DATA_BLOCK "DB_HGU_Execution"
TITLE = 'HGU Execution Variables Data Block'
{ S7_Optimized_Access := 'TRUE' }
VERSION : 1.0
// =============================================================================
// TUSAŞ HGU Control System - Execution Variables Data Block
// TIA Portal S7-1500 Structured Control Language (SCL)
// Generated: 2025-01-14
// Description: All execution variables for HGU system synchronized with UI
// =============================================================================
   VAR
      MOTOR_1_RPM_EXECUTION : Real;   // Motor 1 RPM Execution Value
      MOTOR_1_CURRENT_EXECUTION : Real;   // Motor 1 Current (A) Execution Value
      MOTOR_1_TARGET_EXECUTION : Real;   // Motor 1 Target RPM Execution Value
      MOTOR_1_FLOW_EXECUTION : Real;   // Motor 1 Flow Rate (L/min) Execution Value
      MOTOR_1_PRESSURE_EXECUTION : Real;   // Motor 1 Pressure (bar) Execution Value
      MOTOR_1_LEAK_EXECUTION : Real;   // Motor 1 Leak Rate (L/min) Execution Value
      MOTOR_1_TEMPERATURE_EXECUTION : Real;   // Motor 1 Temperature (°C) Execution Value
      MOTOR_1_STATUS_EXECUTION : USInt;   // Motor 1 Status (0=Offline, 1=Ready, 2=Running, 3=Error)
      MOTOR_1_VALVE_EXECUTION : USInt;   // Motor 1 Valve Control (0=Closed, 1=Open)
      MOTOR_1_LINE_FILTER_EXECUTION : USInt;   // Motor 1 Line Filter Status (0=Error, 1=Warning, 2=OK)
      MOTOR_1_SUCTION_FILTER_EXECUTION : USInt;   // Motor 1 Suction Filter Status (0=Error, 1=OK)
      MOTOR_1_ENABLE_EXECUTION : Bool;   // Motor 1 Enable Control (FALSE=Disabled, TRUE=Enabled)
      MOTOR_1_FLOW_SETPOINT : Real;   // Motor 1 Flow Setpoint (L/min) - User Adjustable from Popup
      // Motor-Pump #2 Variables
      MOTOR_2_RPM_EXECUTION : Real;   // Motor 2 RPM Execution Value
      MOTOR_2_CURRENT_EXECUTION : Real;   // Motor 2 Current (A) Execution Value
      MOTOR_2_TARGET_EXECUTION : Real;   // Motor 2 Target RPM Execution Value
      MOTOR_2_FLOW_EXECUTION : Real;   // Motor 2 Flow Rate (L/min) Execution Value
      MOTOR_2_PRESSURE_EXECUTION : Real;   // Motor 2 Pressure (bar) Execution Value
      MOTOR_2_LEAK_EXECUTION : Real;   // Motor 2 Leak Rate (L/min) Execution Value
      MOTOR_2_TEMPERATURE_EXECUTION : Real;   // Motor 2 Temperature (°C) Execution Value
      MOTOR_2_STATUS_EXECUTION : USInt;   // Motor 2 Status (0=Offline, 1=Ready, 2=Running, 3=Error)
      MOTOR_2_VALVE_EXECUTION : USInt;   // Motor 2 Valve Control (0=Closed, 1=Open)
      MOTOR_2_LINE_FILTER_EXECUTION : USInt;   // Motor 2 Line Filter Status (0=Error, 1=Warning, 2=OK)
      MOTOR_2_SUCTION_FILTER_EXECUTION : USInt;   // Motor 2 Suction Filter Status (0=Error, 1=OK)
      MOTOR_2_ENABLE_EXECUTION : Bool;   // Motor 2 Enable Control (FALSE=Disabled, TRUE=Enabled)
      MOTOR_2_FLOW_SETPOINT : Real;   // Motor 2 Flow Setpoint (L/min) - User Adjustable from Popup
      // Motor-Pump #3 Variables
      MOTOR_3_RPM_EXECUTION : Real;   // Motor 3 RPM Execution Value
      MOTOR_3_CURRENT_EXECUTION : Real;   // Motor 3 Current (A) Execution Value
      MOTOR_3_TARGET_EXECUTION : Real;   // Motor 3 Target RPM Execution Value
      MOTOR_3_FLOW_EXECUTION : Real;   // Motor 3 Flow Rate (L/min) Execution Value
      MOTOR_3_PRESSURE_EXECUTION : Real;   // Motor 3 Pressure (bar) Execution Value
      MOTOR_3_LEAK_EXECUTION : Real;   // Motor 3 Leak Rate (L/min) Execution Value
      MOTOR_3_TEMPERATURE_EXECUTION : Real;   // Motor 3 Temperature (°C) Execution Value
      MOTOR_3_STATUS_EXECUTION : USInt;   // Motor 3 Status (0=Offline, 1=Ready, 2=Running, 3=Error)
      MOTOR_3_VALVE_EXECUTION : USInt;   // Motor 3 Valve Control (0=Closed, 1=Open)
      MOTOR_3_LINE_FILTER_EXECUTION : USInt;   // Motor 3 Line Filter Status (0=Error, 1=Warning, 2=OK)
      MOTOR_3_SUCTION_FILTER_EXECUTION : USInt;   // Motor 3 Suction Filter Status (0=Error, 1=OK)
      MOTOR_3_ENABLE_EXECUTION : Bool;   // Motor 3 Enable Control (FALSE=Disabled, TRUE=Enabled)
      MOTOR_3_FLOW_SETPOINT : Real;   // Motor 3 Flow Setpoint (L/min) - User Adjustable from Popup
      // Motor-Pump #4 Variables
      MOTOR_4_RPM_EXECUTION : Real;   // Motor 4 RPM Execution Value
      MOTOR_4_CURRENT_EXECUTION : Real;   // Motor 4 Current (A) Execution Value
      MOTOR_4_TARGET_EXECUTION : Real;   // Motor 4 Target RPM Execution Value
      MOTOR_4_FLOW_EXECUTION : Real;   // Motor 4 Flow Rate (L/min) Execution Value
      MOTOR_4_PRESSURE_EXECUTION : Real;   // Motor 4 Pressure (bar) Execution Value
      MOTOR_4_LEAK_EXECUTION : Real;   // Motor 4 Leak Rate (L/min) Execution Value
      MOTOR_4_TEMPERATURE_EXECUTION : Real;   // Motor 4 Temperature (°C) Execution Value
      MOTOR_4_STATUS_EXECUTION : USInt;   // Motor 4 Status (0=Offline, 1=Ready, 2=Running, 3=Error)
      MOTOR_4_VALVE_EXECUTION : USInt;   // Motor 4 Valve Control (0=Closed, 1=Open)
      MOTOR_4_LINE_FILTER_EXECUTION : USInt;   // Motor 4 Line Filter Status (0=Error, 1=Warning, 2=OK)
      MOTOR_4_SUCTION_FILTER_EXECUTION : USInt;   // Motor 4 Suction Filter Status (0=Error, 1=OK)
      MOTOR_4_ENABLE_EXECUTION : Bool;   // Motor 4 Enable Control (FALSE=Disabled, TRUE=Enabled)
      MOTOR_4_FLOW_SETPOINT : Real;   // Motor 4 Flow Setpoint (L/min) - User Adjustable from Popup
      // Motor-Pump #5 Variables
      MOTOR_5_RPM_EXECUTION : Real;   // Motor 5 RPM Execution Value
      MOTOR_5_CURRENT_EXECUTION : Real;   // Motor 5 Current (A) Execution Value
      MOTOR_5_TARGET_EXECUTION : Real;   // Motor 5 Target RPM Execution Value
      MOTOR_5_FLOW_EXECUTION : Real;   // Motor 5 Flow Rate (L/min) Execution Value
      MOTOR_5_PRESSURE_EXECUTION : Real;   // Motor 5 Pressure (bar) Execution Value
      MOTOR_5_LEAK_EXECUTION : Real;   // Motor 5 Leak Rate (L/min) Execution Value
      MOTOR_5_TEMPERATURE_EXECUTION : Real;   // Motor 5 Temperature (°C) Execution Value
      MOTOR_5_STATUS_EXECUTION : USInt;   // Motor 5 Status (0=Offline, 1=Ready, 2=Running, 3=Error)
      MOTOR_5_VALVE_EXECUTION : USInt;   // Motor 5 Valve Control (0=Closed, 1=Open)
      MOTOR_5_LINE_FILTER_EXECUTION : USInt;   // Motor 5 Line Filter Status (0=Error, 1=Warning, 2=OK)
      MOTOR_5_SUCTION_FILTER_EXECUTION : USInt;   // Motor 5 Suction Filter Status (0=Error, 1=OK)
      MOTOR_5_ENABLE_EXECUTION : Bool;   // Motor 5 Enable Control (FALSE=Disabled, TRUE=Enabled)
      MOTOR_5_FLOW_SETPOINT : Real;   // Motor 5 Flow Setpoint (L/min) - User Adjustable from Popup
      // Motor-Pump #6 Variables
      MOTOR_6_RPM_EXECUTION : Real;   // Motor 6 RPM Execution Value
      MOTOR_6_CURRENT_EXECUTION : Real;   // Motor 6 Current (A) Execution Value
      MOTOR_6_TARGET_EXECUTION : Real;   // Motor 6 Target RPM Execution Value
      MOTOR_6_FLOW_EXECUTION : Real;   // Motor 6 Flow Rate (L/min) Execution Value
      MOTOR_6_PRESSURE_EXECUTION : Real;   // Motor 6 Pressure (bar) Execution Value
      MOTOR_6_LEAK_EXECUTION : Real;   // Motor 6 Leak Rate (L/min) Execution Value
      MOTOR_6_TEMPERATURE_EXECUTION : Real;   // Motor 6 Temperature (°C) Execution Value
      MOTOR_6_STATUS_EXECUTION : USInt;   // Motor 6 Status (0=Offline, 1=Ready, 2=Running, 3=Error)
      MOTOR_6_VALVE_EXECUTION : USInt;   // Motor 6 Valve Control (0=Closed, 1=Open)
      MOTOR_6_LINE_FILTER_EXECUTION : USInt;   // Motor 6 Line Filter Status (0=Error, 1=Warning, 2=OK)
      MOTOR_6_SUCTION_FILTER_EXECUTION : USInt;   // Motor 6 Suction Filter Status (0=Error, 1=OK)
      MOTOR_6_ENABLE_EXECUTION : Bool;   // Motor 6 Enable Control (FALSE=Disabled, TRUE=Enabled)
      MOTOR_6_FLOW_SETPOINT : Real;   // Motor 6 Flow Setpoint (L/min) - User Adjustable from Popup
      // =============================================================================
      // MOTOR-PUMP #7 VARIABLES (SPECIAL SYSTEM - Different Control Logic)
      // =============================================================================
      MOTOR_7_RPM_EXECUTION : Real;   // Motor 7 RPM (FIXED - Read Only, always 1500 RPM)
      MOTOR_7_CURRENT_EXECUTION : Real;   // Motor 7 Current (A) Execution Value
      MOTOR_7_TARGET_EXECUTION : Real;   // Motor 7 Target RPM (FIXED - Read Only, always 1500 RPM)
      MOTOR_7_FLOW_EXECUTION : Real;   // Motor 7 Flow Rate (FIXED - Read Only, always 34 L/min)
      MOTOR_7_PRESSURE_EXECUTION : Real;   // Motor 7 Pressure (bar) - ADJUSTABLE SETPOINT
      MOTOR_7_LEAK_EXECUTION : Real;   // Motor 7 Leak Rate (L/min) Execution Value
      MOTOR_7_TEMPERATURE_EXECUTION : Real;   // Motor 7 Temperature (°C) Execution Value
      MOTOR_7_STATUS_EXECUTION : USInt;   // Motor 7 Status (0=Offline, 1=Ready, 2=Running, 3=Error)
      MOTOR_7_VALVE_EXECUTION : USInt;   // Motor 7 Valve Control (0=Closed, 1=Open)
      MOTOR_7_LINE_FILTER_EXECUTION : USInt;   // Motor 7 Line Filter Status (0=Error, 1=Warning, 2=OK)
      MOTOR_7_SUCTION_FILTER_EXECUTION : USInt;   // Motor 7 Suction Filter Status (0=Error, 1=OK)
      MOTOR_7_PRESSURE_SETPOINT : Real;   // Motor 7 Pressure Setpoint (bar) - User Adjustable
      MOTOR_7_ENABLE_EXECUTION : Bool;   // Motor 7 Enable Control (FALSE=Disabled, TRUE=Enabled)
      // =============================================================================
      // SYSTEM LEVEL EXECUTION VARIABLES
      // =============================================================================
      // System Control Panel Variables
      SYSTEM_TOTAL_FLOW_EXECUTION : Real;   // Total System Flow Rate (L/min) - Sum of Motor 1-6 flows
      SYSTEM_PRESSURE_EXECUTION : Real;   // System Pressure (bar) - Main system pressure
      SYSTEM_TOTAL_FLOW_SETPOINT : Real;   // Total System Flow Setpoint (L/min) - User Adjustable from Popup
      SYSTEM_PRESSURE_SETPOINT : Real;   // System Pressure Setpoint (bar) - User Adjustable from Popup
      SYSTEM_TANK_LEVEL_EXECUTION : Real;   // Tank Oil Level (%)
      SYSTEM_TANK_TEMPERATURE_EXECUTION : Real;   // Tank Oil Temperature (°C)
      SYSTEM_STATUS_EXECUTION : USInt;   // Overall System Status (0=Offline, 1=Ready, 2=Running, 3=Error, 4=Maintenance)
      // Temperature & Cooling System Variables
      COOLING_AQUA_SENSOR_EXECUTION : Real;   // Aqua/Water Sensor Level (%)
      COOLING_OIL_LEVEL_LITERS_EXECUTION : Real;   // Oil Level in Tank (Liters)
      COOLING_OIL_LEVEL_PERCENT_EXECUTION : Real;   // Oil Level in Tank (%)
      COOLING_OIL_TEMPERATURE_EXECUTION : Real;   // Oil Temperature (°C)
      COOLING_WATER_TEMPERATURE_EXECUTION : Real;   // Water/Coolant Temperature (°C)
      COOLING_SYSTEM_STATUS_EXECUTION : USInt;   // Cooling System Status (0=Offline, 1=Normal, 2=Warning, 3=Critical)
      COOLING_MAX_OIL_TEMP_SETPOINT : Real;   // Maximum Oil Temperature Setpoint (°C) - User Adjustable from Popup
      COOLING_MIN_OIL_TEMP_SETPOINT : Real;   // Minimum Oil Temperature Setpoint (°C) - User Adjustable from Popup
      COOLING_AUTO_CONTROL_ENABLE : Bool;   // Automatic Temperature Control Enable - User Adjustable from Popup
      // System Control Variables
      SYSTEM_CONTROL_MODE_EXECUTION : USInt;   // Control Mode (0=Local, 1=Remote)
      SYSTEM_EMERGENCY_STOP_EXECUTION : Bool;   // Emergency Stop Status (FALSE=Normal, TRUE=Emergency Stop)
      SYSTEM_PUMP_ENABLE_EXECUTION : Bool;   // System Pump Enable (FALSE=Disabled, TRUE=Enabled)
      // Calculated Values (Read-Only)
      TOTAL_ACTIVE_MOTORS : USInt;   // Count of currently running motors
      TOTAL_POWER_CONSUMPTION : Real;   // Total power consumption (kW)
      AVERAGE_SYSTEM_TEMPERATURE : Real;   // Average temperature across all motors
      SYSTEM_EFFICIENCY : Real;   // System efficiency percentage
      // =============================================================================
      // ALARM AND WARNING VARIABLES
      // =============================================================================
      // System Alarms
      ALARM_HIGH_PRESSURE : Bool;   // High Pressure Alarm (FALSE=Normal, TRUE=Alarm)
      ALARM_LOW_PRESSURE : Bool;   // Low Pressure Alarm (FALSE=Normal, TRUE=Alarm)
      ALARM_HIGH_TEMPERATURE : Bool;   // High Temperature Alarm (FALSE=Normal, TRUE=Alarm)
      ALARM_LOW_TANK_LEVEL : Bool;   // Low Tank Level Alarm (FALSE=Normal, TRUE=Alarm)
      ALARM_FILTER_BLOCKED : Bool;   // Filter Blocked Alarm (FALSE=Normal, TRUE=Alarm)
      ALARM_MOTOR_OVERLOAD : Bool;   // Motor Overload Alarm (FALSE=Normal, TRUE=Alarm)
      // Motor Specific Alarm Bitmasks
      MOTOR_ALARM_OVERLOAD_MASK : Byte;   // Motor Overload Alarm Bitmask (bit 0=Motor1, bit 1=Motor2, etc.)
      MOTOR_ALARM_OVERHEAT_MASK : Byte;   // Motor Overheat Alarm Bitmask
      MOTOR_ALARM_LEAK_MASK : Byte;   // Motor Leak Alarm Bitmask

      // =============================================================================
      // SENSOR VARIABLES (From A1.xml - UI Interface)
      // =============================================================================
      Pressure_Supply : Real;   // Main Supply Pressure (0-350 bar) - From A1.xml
      On_Off_Test : Bool;   // Test Signal - From A1.xml
      Pump_Status : Bool;   // Pump Operation Status - From A1.xml
      System_Ready : Bool;   // System Ready Status - From A1.xml
      Temperature_Oil_Tank : Real;   // Tank Oil Temperature (-10 to +80°C) - From A1.xml
      Temperature_Motor : Real;   // Motor Temperature (°C) - From A1.xml
      Pressure_Accumulator : Real;   // Accumulator Pressure (0-350 bar) - From A1.xml

      // =============================================================================
      // MAINTENANCE VARIABLES
      // =============================================================================
      MAINTENANCE_TIMER : Time;   // Maintenance Timer
      LAST_MAINTENANCE_DATE : Date;   // Last Maintenance Date
      NEXT_MAINTENANCE_DUE : Date;   // Next Maintenance Due Date
      AVERAGE_EFFICIENCY : Real;   // Average System Efficiency (%)
      SYSTEM_LOAD_FACTOR : Real;   // System Load Factor (%)
   END_VAR


BEGIN
   MOTOR_1_RPM_EXECUTION := 0.0;
   MOTOR_1_CURRENT_EXECUTION := 0.0;
   MOTOR_1_TARGET_EXECUTION := 0.0;
   MOTOR_1_FLOW_EXECUTION := 0.0;
   MOTOR_1_PRESSURE_EXECUTION := 0.0;
   MOTOR_1_LEAK_EXECUTION := 0.0;
   MOTOR_1_TEMPERATURE_EXECUTION := 0.0;
   MOTOR_1_STATUS_EXECUTION := 0;
   MOTOR_1_VALVE_EXECUTION := 0;
   MOTOR_1_LINE_FILTER_EXECUTION := 0;
   MOTOR_1_SUCTION_FILTER_EXECUTION := 0;
   MOTOR_1_ENABLE_EXECUTION := FALSE;
   MOTOR_1_FLOW_SETPOINT := 45.0;
   MOTOR_2_RPM_EXECUTION := 0.0;
   MOTOR_2_CURRENT_EXECUTION := 0.0;
   MOTOR_2_TARGET_EXECUTION := 0.0;
   MOTOR_2_FLOW_EXECUTION := 0.0;
   MOTOR_2_PRESSURE_EXECUTION := 0.0;
   MOTOR_2_LEAK_EXECUTION := 0.0;
   MOTOR_2_TEMPERATURE_EXECUTION := 0.0;
   MOTOR_2_STATUS_EXECUTION := 0;
   MOTOR_2_VALVE_EXECUTION := 0;
   MOTOR_2_LINE_FILTER_EXECUTION := 0;
   MOTOR_2_SUCTION_FILTER_EXECUTION := 0;
   MOTOR_2_ENABLE_EXECUTION := FALSE;
   MOTOR_2_FLOW_SETPOINT := 32.0;
   MOTOR_3_RPM_EXECUTION := 0.0;
   MOTOR_3_CURRENT_EXECUTION := 0.0;
   MOTOR_3_TARGET_EXECUTION := 0.0;
   MOTOR_3_FLOW_EXECUTION := 0.0;
   MOTOR_3_PRESSURE_EXECUTION := 0.0;
   MOTOR_3_LEAK_EXECUTION := 0.0;
   MOTOR_3_TEMPERATURE_EXECUTION := 0.0;
   MOTOR_3_STATUS_EXECUTION := 0;
   MOTOR_3_VALVE_EXECUTION := 0;
   MOTOR_3_LINE_FILTER_EXECUTION := 0;
   MOTOR_3_SUCTION_FILTER_EXECUTION := 0;
   MOTOR_3_ENABLE_EXECUTION := FALSE;
   MOTOR_3_FLOW_SETPOINT := 32.0;
   MOTOR_4_RPM_EXECUTION := 0.0;
   MOTOR_4_CURRENT_EXECUTION := 0.0;
   MOTOR_4_TARGET_EXECUTION := 0.0;
   MOTOR_4_FLOW_EXECUTION := 0.0;
   MOTOR_4_PRESSURE_EXECUTION := 0.0;
   MOTOR_4_LEAK_EXECUTION := 0.0;
   MOTOR_4_TEMPERATURE_EXECUTION := 0.0;
   MOTOR_4_STATUS_EXECUTION := 0;
   MOTOR_4_VALVE_EXECUTION := 0;
   MOTOR_4_LINE_FILTER_EXECUTION := 0;
   MOTOR_4_SUCTION_FILTER_EXECUTION := 0;
   MOTOR_4_ENABLE_EXECUTION := FALSE;
   MOTOR_4_FLOW_SETPOINT := 38.0;
   MOTOR_5_RPM_EXECUTION := 0.0;
   MOTOR_5_CURRENT_EXECUTION := 0.0;
   MOTOR_5_TARGET_EXECUTION := 0.0;
   MOTOR_5_FLOW_EXECUTION := 0.0;
   MOTOR_5_PRESSURE_EXECUTION := 0.0;
   MOTOR_5_LEAK_EXECUTION := 0.0;
   MOTOR_5_TEMPERATURE_EXECUTION := 0.0;
   MOTOR_5_STATUS_EXECUTION := 0;
   MOTOR_5_VALVE_EXECUTION := 0;
   MOTOR_5_LINE_FILTER_EXECUTION := 0;
   MOTOR_5_SUCTION_FILTER_EXECUTION := 0;
   MOTOR_5_ENABLE_EXECUTION := FALSE;
   MOTOR_5_FLOW_SETPOINT := 25.0;
   MOTOR_6_RPM_EXECUTION := 0.0;
   MOTOR_6_CURRENT_EXECUTION := 0.0;
   MOTOR_6_TARGET_EXECUTION := 0.0;
   MOTOR_6_FLOW_EXECUTION := 0.0;
   MOTOR_6_PRESSURE_EXECUTION := 0.0;
   MOTOR_6_LEAK_EXECUTION := 0.0;
   MOTOR_6_TEMPERATURE_EXECUTION := 0.0;
   MOTOR_6_STATUS_EXECUTION := 0;
   MOTOR_6_VALVE_EXECUTION := 0;
   MOTOR_6_LINE_FILTER_EXECUTION := 0;
   MOTOR_6_SUCTION_FILTER_EXECUTION := 0;
   MOTOR_6_ENABLE_EXECUTION := FALSE;
   MOTOR_6_FLOW_SETPOINT := 40.0;
   MOTOR_7_RPM_EXECUTION := 1500.0;
   MOTOR_7_CURRENT_EXECUTION := 0.0;
   MOTOR_7_TARGET_EXECUTION := 1500.0;
   MOTOR_7_FLOW_EXECUTION := 34.0;
   MOTOR_7_PRESSURE_EXECUTION := 0.0;
   MOTOR_7_LEAK_EXECUTION := 0.0;
   MOTOR_7_TEMPERATURE_EXECUTION := 0.0;
   MOTOR_7_STATUS_EXECUTION := 0;
   MOTOR_7_VALVE_EXECUTION := 0;
   MOTOR_7_LINE_FILTER_EXECUTION := 0;
   MOTOR_7_SUCTION_FILTER_EXECUTION := 0;
   MOTOR_7_PRESSURE_SETPOINT := 250.0;
   MOTOR_7_ENABLE_EXECUTION := FALSE;
   SYSTEM_TOTAL_FLOW_EXECUTION := 0.0;
   SYSTEM_PRESSURE_EXECUTION := 0.0;
   SYSTEM_TOTAL_FLOW_SETPOINT := 180.0;
   SYSTEM_PRESSURE_SETPOINT := 280.0;
   SYSTEM_TANK_LEVEL_EXECUTION := 0.0;
   SYSTEM_TANK_TEMPERATURE_EXECUTION := 0.0;
   SYSTEM_STATUS_EXECUTION := 0;
   COOLING_AQUA_SENSOR_EXECUTION := 0.0;
   COOLING_OIL_LEVEL_LITERS_EXECUTION := 0.0;
   COOLING_OIL_LEVEL_PERCENT_EXECUTION := 0.0;
   COOLING_OIL_TEMPERATURE_EXECUTION := 0.0;
   COOLING_WATER_TEMPERATURE_EXECUTION := 0.0;
   COOLING_SYSTEM_STATUS_EXECUTION := 0;
   COOLING_MAX_OIL_TEMP_SETPOINT := 55.0;
   COOLING_MIN_OIL_TEMP_SETPOINT := 40.0;
   COOLING_AUTO_CONTROL_ENABLE := TRUE;
   SYSTEM_CONTROL_MODE_EXECUTION := 0;
   SYSTEM_EMERGENCY_STOP_EXECUTION := FALSE;
   SYSTEM_PUMP_ENABLE_EXECUTION := FALSE;
   TOTAL_ACTIVE_MOTORS := 0;
   TOTAL_POWER_CONSUMPTION := 0.0;
   AVERAGE_SYSTEM_TEMPERATURE := 0.0;
   SYSTEM_EFFICIENCY := 0.0;
   ALARM_HIGH_PRESSURE := FALSE;
   ALARM_LOW_PRESSURE := FALSE;
   ALARM_HIGH_TEMPERATURE := FALSE;
   ALARM_LOW_TANK_LEVEL := FALSE;
   ALARM_FILTER_BLOCKED := FALSE;
   ALARM_MOTOR_OVERLOAD := FALSE;
   MOTOR_ALARM_OVERLOAD_MASK := 16#00;
   MOTOR_ALARM_OVERHEAT_MASK := 16#00;
   MOTOR_ALARM_LEAK_MASK := 16#00;

   // Initialize A1.xml sensor variables
   Pressure_Supply := 0.0;
   On_Off_Test := FALSE;
   Pump_Status := FALSE;
   System_Ready := FALSE;
   Temperature_Oil_Tank := 0.0;
   Temperature_Motor := 0.0;
   Pressure_Accumulator := 0.0;

   // Initialize maintenance variables
   MAINTENANCE_TIMER := T#0MS;
   LAST_MAINTENANCE_DATE := D#1990-01-01;
   NEXT_MAINTENANCE_DUE := D#1990-01-01;
   AVERAGE_EFFICIENCY := 0.0;
   SYSTEM_LOAD_FACTOR := 0.0;

END_DATA_BLOCK